FUNCTION_BLOCK PY_MQTT_PUB (* MQTT Publisher FB for Dinasore *)
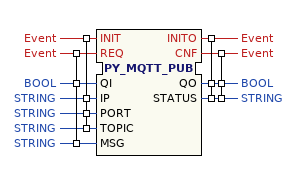
  EVENT_INPUT
    INIT WITH PORT, TOPIC, IP;
    REQ WITH QI, MSG;
  END_EVENT
  EVENT_OUTPUT
    INITO WITH QO, STATUS;
    CNF WITH STATUS, QO;
  END_EVENT
  VAR_INPUT
    QI : BOOL;
    IP : STRING;
    PORT : STRING;
    TOPIC : STRING;
    MSG : STRING;
  END_VAR
  VAR_OUTPUT
    QO : BOOL;
    STATUS : STRING;
  END_VAR
END_FUNCTION_BLOCK
